% RSLogix 500 project FULL ADDER 2.RSS, saved by version 8.30.00.15 %
PROJECT "UNTITLED"    % processor: MicroLogix 1000 %

PROGRAM FILES
  LAD 2 "MAIN_PROG"  4 rungs
  LAD 3 "USER_FAULT"  1 rungs
  LAD 4 "HSC_INT"  1 rungs
  LAD 5 "STI_INT"  1 rungs
  LAD 6, 7, 8, 9, 10, 11, 12, 13, 14, 15, 16: only END

DATA FILES
  O0 OUTPUT  1 elements
  I1 INPUT  2 elements
  S2 STATUS  33 elements
  B3 BINARY  32 elements
  T4 TIMER  40 elements
  C5 COUNTER  32 elements
  R6 CONTROL  16 elements
  N7 INTEGER  105 elements

LADDER 2 "MAIN_PROG"
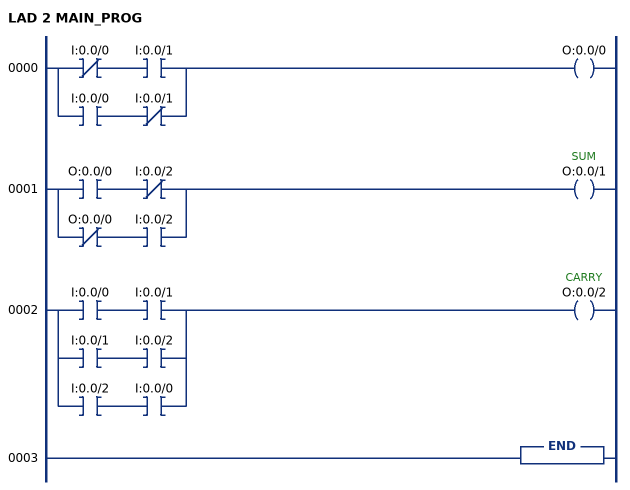
% Rung: 0 %
SOR BST XIO I:0.0/0 XIC I:0.0/1 NXB XIC I:0.0/0 XIO I:0.0/1 BND OTE O:0.0/0 EOR
% Rung: 1 %
SOR BST XIC O:0.0/0 XIO I:0.0/2 NXB XIO O:0.0/0 XIC I:0.0/2 BND OTE O:0.0/1 EOR
%   O:0.0/1  "SUM" %
% Rung: 2 %
SOR BST BST XIC I:0.0/0 XIC I:0.0/1 NXB XIC I:0.0/1 XIC I:0.0/2 BND NXB XIC I:0.0/2 XIC I:0.0/0 BND OTE O:0.0/2 EOR
%   O:0.0/2  "CARRY" %
% Rung: 3 %
SOR END EOR
